TYPE CoE_Obj_typ :
STRUCT
	Index  	 : WORD;
	SunIndex : BYTE;
	Size	 : UDINT;   
	IsReal 	 : BOOL;  

END_STRUCT
END_TYPE

(* stored: Version 1.1.0.1, ProductVersion 3.1.4024.3
   DUT CoE_Obj_typ: Id {6e088ad0-f329-0add-05fd-c76160fb18ce} *)
